TYPE COMPLEX :
STRUCT
	re : REAL;
	im : REAL;
END_STRUCT
END_TYPE

(* stored: Version 1.1.0.1, ProductVersion 3.1.4022.7
   DUT COMPLEX: Id {674666fb-7a14-4e39-a3d2-7dd5e5adcec8} *)
